// TIA Portal V19 export
FUNCTION_BLOCK "PTrkMng_FB"   // FB176, LAD
// stored: MemoryReserve 100, SetENOAutomatically false
   VAR_INPUT
      Area : "AreaInterface";
      A0202_MotionStandstill : Bool;
   END_VAR
   VAR CONSTANT
      HMI_COLOR_LIGHT_GREY : Int := 0;
      HMI_COLOR_DARK_GREY : Int := 1;
      HMI_COLOR_RED : Int := 2;
      HMI_COLOR_GREEN : Int := 3;
   END_VAR
   VAR_TEMP   // added for the SCL form of the ladder/FBD networks
      _w1 : Bool;
      _w2 : Bool;
   END_VAR
BEGIN

REGION Network 1: HMI - Gestione ricondizionamento
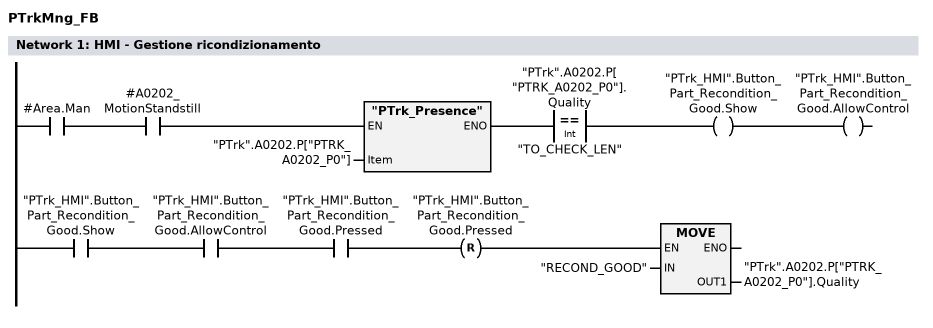
   RUNG wire#powerrail
      Contact( #Area.Man )
      Contact( #A0202_MotionStandstill )
      "PTrk_Presence"(Item := "PTrk".A0202.P["PTRK_A0202_P0"])
      { S7_Templates := "SrcType := Int" } EQ_Contact(in1 := "PTrk".A0202.P["PTRK_A0202_P0"].Quality, in2 := "TO_CHECK_LEN")
      Coil( "PTrk_HMI".Button_Part_Recondition_Good.Show )
      Coil( "PTrk_HMI".Button_Part_Recondition_Good.AllowControl )
   END_RUNG
   RUNG wire#powerrail
      Contact( "PTrk_HMI".Button_Part_Recondition_Good.Show )
      Contact( "PTrk_HMI".Button_Part_Recondition_Good.AllowControl )
      Contact( "PTrk_HMI".Button_Part_Recondition_Good.Pressed )
      R_Coil( "PTrk_HMI".Button_Part_Recondition_Good.Pressed )
      Move(in := "RECOND_GOOD", out1 => "PTrk".A0202.P["PTRK_A0202_P0"].Quality)
   END_RUNG
   // the same network as SCL:
   "PTrk_Presence"(EN := #Area.Man AND #A0202_MotionStandstill,
                   Item := "PTrk".A0202.P["PTRK_A0202_P0"],
                   ENO => #_w1);
   "PTrk_HMI".Button_Part_Recondition_Good.Show := #_w1 AND ("PTrk".A0202.P["PTRK_A0202_P0"].Quality = "TO_CHECK_LEN");
   "PTrk_HMI".Button_Part_Recondition_Good.AllowControl := "PTrk_HMI".Button_Part_Recondition_Good.Show;
   #_w2 := "PTrk_HMI".Button_Part_Recondition_Good.Show AND "PTrk_HMI".Button_Part_Recondition_Good.AllowControl AND "PTrk_HMI".Button_Part_Recondition_Good.Pressed;
   IF #_w2 THEN
       "PTrk_HMI".Button_Part_Recondition_Good.Pressed := FALSE;
       "PTrk".A0202.P["PTRK_A0202_P0"].Quality := "RECOND_GOOD";
   END_IF;
END_REGION
END_FUNCTION_BLOCK
